// TIA Portal V18 export
FUNCTION_BLOCK "Process"   // FB1, LAD
VERSION : 0.1
// stored: Access Unpublished, AutoNumber true, IsIECCheckEnabled false, IsRetainMemResEnabled false, MemoryReserve 100, Namespace Coagulation, SetENOAutomatically false, UDAEnableTagReadback false
BEGIN
END_FUNCTION_BLOCK
